TYPE T_QueryInterface : __SYSTEM.IQueryInterface; END_TYPE

(* stored: Version 1.1.0.1
   DUT T_QueryInterface: Id {ebd27d8f-dbc2-0d7b-240c-1789cde44b12} *)
